Fanuc KAREL source: VT_GET_AREID.kl

PROGRAM T
%NOLOCKGROUP
VAR
 v0 : STRING[40]
 res : INTEGER
BEGIN
 res = VT_GET_AREID(v0)
END T
